(* CODESYS project Eurowin_v_1_1Test.project

Project tree, tasks and I/O mapping:
  Device : CODESYS Control Win V3, 3S - Smart Software Solutions GmbH, order no. 305021, version 3.5.5.50
    application Application
      libraries: Standard, * (System); Util, * (System); Mx110Assistant, 3.5.4.0 (Owen)
      task MainTask (cyclic, interval t#10ms, priority 1) calls PLC_PRG
      task VISU_TASK (cyclic, interval 100 ms, priority 31) calls VisuElems.Visu_Prg
      program PLC_PRG [ST]: incrSpeed, decrSpeed, init, valveWork, lamp1Work, getData, setData
      visualisation Main
      visualisation Alarm
      visualisation TestParameters
      image pool ImagePool
    Modbus_COM : Modbus COM, 3S - Smart Software Solutions GmbH, version 3.4.0.0
        settings: DataBits = 8; StopBits = 1; ComPort = 2
      Modbus_Master_COM_Port : Modbus Master, COM Port, 3S - Smart Software Solutions GmbH, version 3.5.5.0
          settings: Transmission = 'RTU'; ResponseTimeout = 300; TimeBetweenFrames = 10; Auto-restart communication = TRUE
        MU110_8I : MU110-8I, Owen, order no. 3.5.4.2, version 3.5.4.0
            settings: SlaveAddress = 1; ResponseTimeout = 300; UseExtendedFunctionCodes = TRUE
            unmapped channels: r.OE_1, in1, out1
        MV110_8A : MV110-8A, Owen, order no. 3.5.4.8, version 3.5.4.0
            settings: SlaveAddress = 17; ResponseTimeout = 300; UseExtendedFunctionCodes = TRUE
            unmapped channels: DP_1, in1, out1
        MU110_16R_K : MU110-16R_K, Owen, order no. 3.5.4.2, version 3.5.4.0
            settings: SlaveAddress = 33; ResponseTimeout = 300; UseExtendedFunctionCodes = TRUE
            unmapped channels: rMask, wMask, in1, out1
  text list GlobalTextList
  5ce3da45-db07-42e7-a21c-a00fff4ed8f6|D:\Pictures\ICONS\OnOff\off.png
  5ce3da45-db07-42e7-a21c-a00fff4ed8f6|D:\Pictures\ICONS\OnOff\on.png
*)

// Device/Application/PLC_PRG
PROGRAM PLC_PRG
VAR
	tmr1:TON;
	tpValve1:TP;
	blValve:BLINK;
	
	iMaxSpeed:INT := 14;
	iMinSpeed:INT := 1;
	bInit:BOOL := TRUE;
	
	sTime:STRING;
	iIn, iOut, iUst, iSpeed :INT;
	bRun, bRunAuto, bLamp1, bLamp2, bKlap1, bKlap2, bKlap3, bKlap4, bInLevel:BOOL;
	rTemp1, rTemp2, rTemp3 : REAL;
END_VAR

init();

getData();

valveWork();
lamp1Work();

setData();

ACTION incrSpeed:
IF iSpeed < iMaxSpeed THEN
	iSpeed := iSpeed + 1;
END_IF
END_ACTION

ACTION decrSpeed:
IF iSpeed > iMinSpeed THEN
	iSpeed := iSpeed - 1;
END_IF
END_ACTION

ACTION init:
IF bInit THEN
	iSpeed := 1;
	bInit := FALSE;
END_IF
END_ACTION

ACTION valveWork:
IF bRun THEN
	blValve(ENABLE := bRun, TIMEHIGH := INT_TO_TIME(1000 * iSpeed), TIMELOW := INT_TO_TIME(1000));
	bKlap1 := blValve.OUT AND blValve.ENABLE;
	bKlap2 := blValve.OUT AND blValve.ENABLE;
	bKlap3 := blValve.OUT AND blValve.ENABLE;
	bKlap4 := blValve.OUT AND blValve.ENABLE;
	bRunAuto := TRUE;
END_IF
IF bRunAuto AND NOT bRun THEN
	bKlap1 := FALSE;
	bKlap2 := FALSE;
	bKlap3 := FALSE;
	bKlap4 := FALSE;
	bRunAuto := FALSE;
END_IF
END_ACTION

ACTION lamp1Work:
IF iIn < iUst THEN
	bLamp1 := TRUE;
	tmr1(IN := FALSE);
ELSE
	tmr1(IN := TRUE, PT := T#5S);
	bLamp1 := NOT tmr1.Q;
	sTime := TIME_TO_STRING(tmr1.PT - tmr1.ET);
END_IF
END_ACTION

ACTION getData:
rTemp1 := MV110_8A.rEAd_1;
rTemp2 := MV110_8A.rEAd_2;
rTemp3 := MV110_8A.rEAd_3;
END_ACTION

ACTION setData:

END_ACTION

END_PROGRAM

// Device/Application/Main
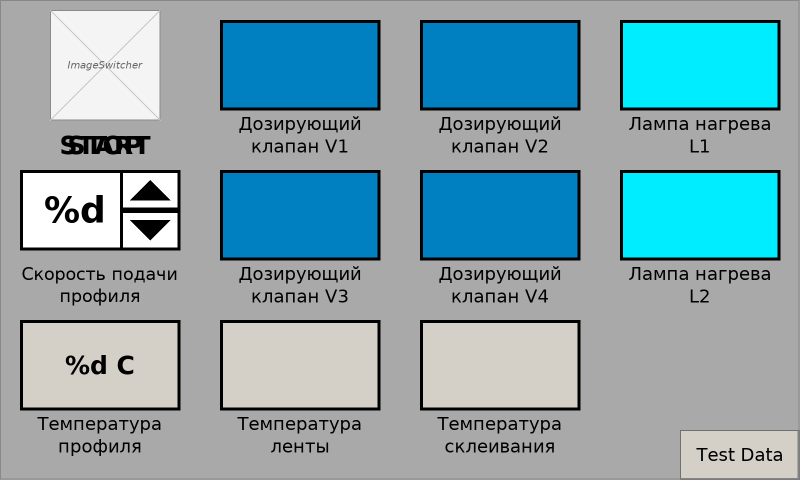
VISUALIZATION Main  // 800x480
    RoundedRectangle (620,20 160x90), colour toggle: PLC_PRG.bLamp1
    RoundedRectangle (620,170 160x90)
    RoundedRectangle (20,170 110x80), "%d", text variable: PLC_PRG.iSpeed
    RoundedRectangle (220,20 160x90), colour toggle: PLC_PRG.bKlap1
        OnMouseClick:  ToggleVariable=PLC_PRG.bKlap1
    RoundedRectangle (20,320 160x90), "%d C", text variable: PLC_PRG.iIn
    RoundedRectangle (220,320 160x90)
    RoundedRectangle (420,320 160x90)
    RoundedRectangle (20,260 160x50), "Скорость подачи профиля"
    RoundedRectangle (220,110 160x50), "Дозирующий клапан V1"
    RoundedRectangle (420,110 160x50), "Дозирующий клапан V2"
    RoundedRectangle (220,260 160x50), "Дозирующий клапан V3"
    RoundedRectangle (420,260 160x50), "Дозирующий клапан V4"
    RoundedRectangle (620,110 160x50), "Лампа нагрева L1"
    RoundedRectangle (620,260 160x50), "Лампа нагрева L2"
    RoundedRectangle (20,410 160x50), "Температура профиля"
    RoundedRectangle (220,410 160x50), "Температура ленты"
    RoundedRectangle (420,410 160x50), "Температура склеивания"
    RoundedRectangle (120,170 60x40)
        OnMouseClick: execute { PLC_PRG.incrSpeed(); }
    RoundedRectangle (120,210 60x40)
        OnMouseClick: execute { PLC_PRG.decrSpeed(); }
    Polygon (130,200) (150,180) (170,200)
        OnMouseClick: execute { PLC_PRG.incrSpeed(); }
    Polygon (130,220) (150,240) (170,220)
        OnMouseClick: execute { PLC_PRG.decrSpeed(); }
    RoundedRectangle (420,20 160x90), colour toggle: PLC_PRG.bKlap2
        OnMouseClick:  ToggleVariable=PLC_PRG.bKlap2
    RoundedRectangle (220,170 160x90), colour toggle: PLC_PRG.bKlap3
        OnMouseClick:  ToggleVariable=PLC_PRG.bKlap3
    RoundedRectangle (420,170 160x90), colour toggle: PLC_PRG.bKlap4
        OnMouseClick:  ToggleVariable=PLC_PRG.bKlap4
    RoundedRectangle (30,120 150x50), "START", invisible if: PLC_PRG.bRun
    ImageSwitcher (50,10 110x110), variable: PLC_PRG.bRun, background image: ImagePool.off, image: ImagePool.on, behaviour: TOGGLE
    RoundedRectangle (30,120 150x50), "STOP", invisible if: NOT PLC_PRG.bRun
    Button (680,430 120x50), "Test Data"
        OnMouseClick:  Assign=TestParameters, Type=Assignment
END_VISUALIZATION

// Device/Application/Alarm
VISUALIZATION Alarm  // 800x480
END_VISUALIZATION

// Device/Application/TestParameters
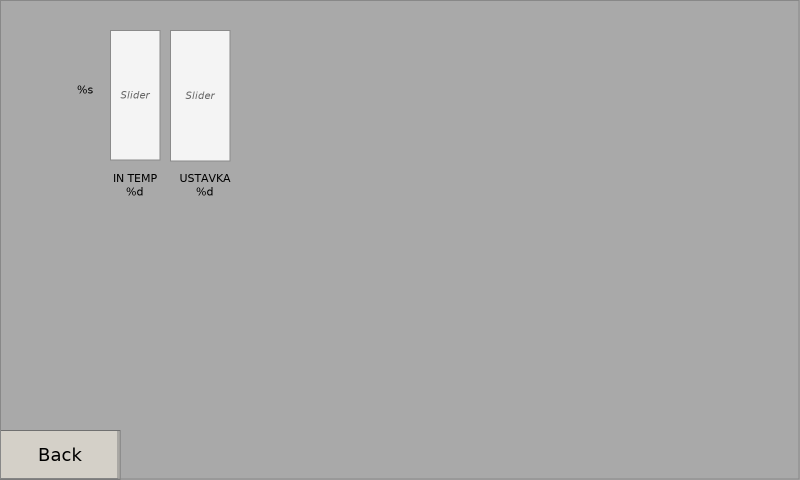
VISUALIZATION TestParameters  // 800x480
    RoundedRectangle (170,170 70x30), "USTAVKA %d", text variable: PLC_PRG.iUst
    Slider (110,30 50x130), variable: PLC_PRG.iIn, scale 0..100
    Slider (170,30 60x131), variable: PLC_PRG.iUst, scale 0..100
    RoundedRectangle (100,170 70x30), "IN TEMP %d", text variable: PLC_PRG.iIn
    RoundedRectangle (50,70 70x40), "%s", text variable: PLC_PRG.sTime
    Button (0,430 120x50), "Back"
        OnMouseClick:  Assign=Main, Type=Assignment
END_VISUALIZATION
